Staubli VAL3: T2.dtx

public frame fReference = {x=1300, y=217.412, z=-659.53, rz=90, fatherId=world[0]}
public jointRx jPark = {j3=90, j5=90}
public jointRx jJoint = {j1=0.76736, j2=38.58214, j3=106.5226, j5=34.89526, j6=90.76736}
public mdesc mNomSpeed = {blend=off}
public mdesc mSpeed[12]
  [0] = {tmax=30, rmax=100, leave=0.1, reach=0.1, blend=cartesian}
  [1] = {tmax=30, rmax=100, leave=0.1, reach=0.1, blend=cartesian}
  [2] = {tmax=30, rmax=100, leave=0.1, reach=0.1, blend=cartesian}
  [3] = {tmax=30, rmax=100, leave=0.1, reach=0.1, blend=cartesian}
  [4] = {tmax=30, rmax=100, leave=0.1, reach=0.1, blend=cartesian}
  [5] = {tmax=30, rmax=100, leave=0.1, reach=0.1, blend=cartesian}
  [6] = {tmax=30, rmax=100, leave=0.1, reach=0.1, blend=cartesian}
  [7] = {tmax=30, rmax=100, leave=0.1, reach=0.1, blend=cartesian}
  [8] = {tmax=30, rmax=100, leave=0.1, reach=0.1, blend=cartesian}
  [9] = {tmax=30, rmax=100, leave=0.1, reach=0.1, blend=cartesian}
  [10] = {tmax=30, rmax=100, leave=0.1, reach=0.1, blend=cartesian}
  [11] = {tmax=30, rmax=100, leave=0.1, reach=0.1, blend=cartesian}
public num nTraj
num nTimeStop
num nTimeStart
num nMode
num nEtat
public pointRx pPoint[40]
  [0] = {x=-200, z=100, rx=-180, shoulder=lefty, elbow=epositive, wrist=wpositive, fatherId=fReference[0]}
  [1] = {x=-200, rx=180, shoulder=lefty, elbow=epositive, wrist=wpositive, fatherId=fReference[0]}
  [2] = {x=-200, rx=180, shoulder=lefty, elbow=epositive, wrist=wpositive, fatherId=fReference[0]}
  [3] = {x=-120, rx=-180, shoulder=lefty, elbow=epositive, wrist=wpositive, fatherId=fReference[0]}
  [4] = {x=-40, rx=180, shoulder=lefty, elbow=epositive, wrist=wpositive, fatherId=fReference[0]}
  [5] = {x=40, rx=180, shoulder=lefty, elbow=epositive, wrist=wpositive, fatherId=fReference[0]}
  [6] = {x=120, rx=-180, shoulder=lefty, elbow=epositive, wrist=wpositive, fatherId=fReference[0]}
  [7] = {x=200, rx=180, shoulder=lefty, elbow=epositive, wrist=wpositive, fatherId=fReference[0]}
  [8] = {x=200, rx=180, shoulder=lefty, elbow=epositive, wrist=wpositive, fatherId=fReference[0]}
  [9] = {x=200, z=100, rx=-180, rz=-179.277, shoulder=lefty, elbow=epositive, wrist=wpositive, fatherId=fReference[0]}
  [10] = {y=-22, z=100, rx=-180, rz=173.723, shoulder=lefty, elbow=epositive, wrist=wpositive, fatherId=fReference[0]}
  [11] = {y=-22, rx=180, rz=173.723, shoulder=lefty, elbow=epositive, wrist=wpositive, fatherId=fReference[0]}
  [12] = {y=-22, rx=-180, rz=90, shoulder=lefty, elbow=epositive, wrist=wpositive, fatherId=fReference[0]}
  [13] = {y=-102, rx=-180, rz=90, shoulder=lefty, elbow=epositive, wrist=wpositive, fatherId=fReference[0]}
  [14] = {y=-182, rx=-180, rz=90, shoulder=lefty, elbow=epositive, wrist=wpositive, fatherId=fReference[0]}
  [15] = {y=-262, rx=-180, rz=90, shoulder=lefty, elbow=epositive, wrist=wpositive, fatherId=fReference[0]}
  [16] = {y=-342, rx=-180, rz=90, shoulder=lefty, elbow=epositive, wrist=wpositive, fatherId=fReference[0]}
  [17] = {y=-422, rx=-180, rz=90, shoulder=lefty, elbow=epositive, wrist=wpositive, fatherId=fReference[0]}
  [18] = {y=-422, rx=-180, rz=90, shoulder=lefty, elbow=epositive, wrist=wpositive, fatherId=fReference[0]}
  [19] = {y=-422, z=100, rx=-180, rz=90, shoulder=lefty, elbow=epositive, wrist=wpositive, fatherId=fReference[0]}
  [20] = {y=-422, z=122, rx=-180, rz=90, shoulder=lefty, elbow=epositive, wrist=wpositive, fatherId=fReference[0]}
  [21] = {y=-422, z=22, rx=-180, rz=90, shoulder=lefty, elbow=epositive, wrist=wpositive, fatherId=fReference[0]}
  [22] = {y=-422, z=22, rx=180, rz=-90, shoulder=lefty, elbow=epositive, wrist=wpositive, fatherId=fReference[0]}
  [23] = {y=-342, z=22, rx=180, rz=-90, shoulder=lefty, elbow=epositive, wrist=wpositive, fatherId=fReference[0]}
  [24] = {y=-262, z=22, rx=180, rz=-90, shoulder=lefty, elbow=epositive, wrist=wpositive, fatherId=fReference[0]}
  [25] = {y=-182, z=22, rx=180, rz=-90, shoulder=lefty, elbow=epositive, wrist=wpositive, fatherId=fReference[0]}
  [26] = {y=-102, z=22, rx=180, rz=-90, shoulder=lefty, elbow=epositive, wrist=wpositive, fatherId=fReference[0]}
  [27] = {y=-22, z=22, rx=180, rz=-90, shoulder=lefty, elbow=epositive, wrist=wpositive, fatherId=fReference[0]}
  [28] = {y=-22, z=22, rx=180, rz=-90, shoulder=lefty, elbow=epositive, wrist=wpositive, fatherId=fReference[0]}
  [29] = {y=-22, z=122, rx=-180, rz=-173.723, shoulder=lefty, elbow=epositive, wrist=wpositive, fatherId=fReference[0]}
  [30] = {x=-200, z=122, rx=-180, rz=-173.723, shoulder=lefty, elbow=epositive, wrist=wpositive, fatherId=fReference[0]}
  [31] = {x=-200, z=22, rx=-180, rz=-173.723, shoulder=lefty, elbow=epositive, wrist=wpositive, fatherId=fReference[0]}
  [32] = {x=-200, z=22, rx=-180, shoulder=lefty, elbow=epositive, wrist=wpositive, fatherId=fReference[0]}
  [33] = {x=-120, z=22, rx=180, shoulder=lefty, elbow=epositive, wrist=wpositive, fatherId=fReference[0]}
  [34] = {x=-40, z=22, rx=-180, shoulder=lefty, elbow=epositive, wrist=wpositive, fatherId=fReference[0]}
  [35] = {x=40, z=22, rx=180, shoulder=lefty, elbow=epositive, wrist=wpositive, fatherId=fReference[0]}
  [36] = {x=120, z=22, rx=-180, shoulder=lefty, elbow=epositive, wrist=wpositive, fatherId=fReference[0]}
  [37] = {x=200, z=22, rx=-180, shoulder=lefty, elbow=epositive, wrist=wpositive, fatherId=fReference[0]}
  [38] = {x=200, z=22, rx=-180, shoulder=lefty, elbow=epositive, wrist=wpositive, fatherId=fReference[0]}
  [39] = {x=200, z=122, rx=180, shoulder=lefty, elbow=epositive, wrist=wpositive, fatherId=fReference[0]}
public tool tTool = {z=452, fatherId=flange[0], ioLink=valve1}
dio doValve1 = {link=valve1}
aio Tpompe = {link=CanIO\RemIO\remio0_QW}
